FUNCTION_BLOCK "FB_Machine_Spinner"
{ S7_Optimized_Access := 'TRUE' }
VERSION : 0.1
   VAR_INPUT
      Enable : Bool;
      MC_number : Int;
      MC_inRemoteMode : Bool;
      AutoModeFromHandController : Bool;
   END_VAR

   VAR_IN_OUT
      io_in : "UDT_MachineIn";
      io_out : "UDT_MachineOut";
      Status : Int;
      Mode : "UDT_MachineMode";
      cmd : "UDT_CMD";
      order : "UDT_Order";
      pallet : Int;
      fixture : Int;
      ManualVice : Int;
      piecepresent : Array[1..5] of Int;
      viceLocked : Bool;
      viceUnlocked : Bool;
      palletLocked : Bool;
      changePalletReq : Bool;
      lastMission : Int;
      Dispatcher : Array[0..10] of Int;
      subState : Int;
      autoModePrev : Bool;
   END_VAR

   VAR
      "timer" {InstructionName := 'TON_TIME'; LibVersion := '1.0'; S7_SetPoint := 'False'} : Array[0..10] of TON_TIME;
      queryTemp { S7_SetPoint := 'True'} : String;
      doorOpened : Bool;
      enablePrev : Bool;
   END_VAR

   VAR_TEMP
      timeout : Time;
      i : Int;
      countPieces : Int;
      oldStatus : Int;
      tmpUint : UInt;
      Dispatcher_old : Array[0..10] of Int;
   END_VAR


BEGIN
	REGION ENABLE_GATE
	    // Azzero le uscite UNA VOLTA SOLA (fronte di disable) e RETURN.
	    // io_out e' condiviso tra le istanze dei tipi: azzerare a ogni scan
	    // cancellerebbe le uscite mantenute del tipo ATTIVO.
	    IF NOT #Enable THEN
	        IF #enablePrev THEN
	            #io_out.openDoor := FALSE;
	            #io_out.closeDoor := FALSE;
	            #io_out.openVice := FALSE;
	            #io_out.closeVice := FALSE;
	            #io_out.unlockPallet := FALSE;
	            #io_out.lockPallet := FALSE;
	            #io_out.unlockPartOnTable := FALSE;
	            #io_out.lockPartOnTable := FALSE;
	            #io_out.startWork := FALSE;
	            #io_out.startWash := FALSE;
	            #io_out.fuoriIngombro := FALSE;
	        END_IF;
	        #enablePrev := FALSE;
	        RETURN;
	    END_IF;
	    #enablePrev := TRUE;
	END_REGION

	REGION GENERIC_implementation

	    #countPieces := 0;
	    FOR #i := 1 TO 5 DO
	        IF #piecepresent[#i] > 0 THEN
	            #countPieces := #countPieces + 1;
	        END_IF;
	    END_FOR;

	    #oldStatus := #Status;
	    IF #countPieces = 0 THEN
	        IF #pallet = 0 AND #ManualVice = 0 THEN
	            #Status := DINT_TO_INT("UNLOADED");     // totally empty machine
	        ELSE
	            #Status := DINT_TO_INT("EMPTY");        // pallet and fixture mounted on machine but not one piece inside
	        END_IF;

	    ELSIF "DB_Robot".MissionCode = 0 AND #lastMission = "MISSION_LoadPallet_MC" THEN
	        #Status := DINT_TO_INT("EMPTY");
	        #lastMission := 0;

	    ELSIF "DB_Robot".MissionCode = 0 AND #lastMission = "MISSION_UnloadPallet_MC" THEN
	        #Status := DINT_TO_INT("UNLOADED");
	        #lastMission := 0;

	    ELSIF "DB_Robot".MissionCode = 0 AND #lastMission = "MISSION_LoadManVice" THEN
	        #Status := DINT_TO_INT("EMPTY");
	        #lastMission := 0;

	    ELSIF "DB_Robot".MissionCode = 0 AND #lastMission = "MISSION_UnloadManVice" THEN
	        #Status := DINT_TO_INT("UNLOADED");
	        #lastMission := 0;

	    ELSIF FIND(IN1 := "DB_MQTT".lastTopicReceived, IN2 := 'MC1') >= 0 AND #MC_number = 1 THEN  //EG: MC1/CHANGEPALLET
	        IF FIND(IN1 := "DB_MQTT".lastTopicReceived, IN2 := 'CHANGEPALLET') >= 0 THEN
	            #changePalletReq := ("DB_MQTT".lastCmdReceived = 1);
	        ELSIF FIND(IN1 := "DB_MQTT".lastTopicReceived, IN2 := 'CN_STATUS') >= 0 THEN
	            #Status := "DB_MQTT".lastCmdReceived;
	        END_IF;

	    ELSIF FIND(IN1 := "DB_MQTT".lastTopicReceived, IN2 := 'MC2') >= 0 AND #MC_number = 2 THEN  //EG: MC2/CHANGEPALLET
	        IF FIND(IN1 := "DB_MQTT".lastTopicReceived, IN2 := 'CHANGEPALLET') >= 0 THEN
	            #changePalletReq := ("DB_MQTT".lastCmdReceived = 1);
	        ELSIF FIND(IN1 := "DB_MQTT".lastTopicReceived, IN2 := 'CN_STATUS') >= 0 THEN
	            #Status := "DB_MQTT".lastCmdReceived;
	        END_IF;
	    END_IF;

	    IF (#Status >= 0 AND (#Status <> #oldStatus)) THEN
	        "FC_MQTT"(insert := true,
	                  send := false,
	                  topic := CONCAT(IN1 := 'FROM_PLANT/STATUS/MC', IN2 := "INT_TO_STRING_WITHOUT_SIGN"(#MC_number)),
	                  payload := STRING_TO_WSTRING("INT_TO_STRING_WITHOUT_SIGN"(#Status)));
	        #oldStatus := #Status;
	    END_IF;

	END_REGION ;

	FOR #i := 0 TO 10 DO
	    #Dispatcher_old[#i] := #Dispatcher[#i];
	END_FOR;

	REGION Manager CMD from HMI
	    // i comandi HMI non devono interferire col dispatcher
	    IF "DB_MQTT".lastTopicReceived = CONCAT_STRING(IN1 := 'MC', IN2 := "INT_TO_STRING_WITHOUT_SIGN"(#MC_number))
	        AND "DB_RobotMissionStatus".StatusCode = "cmd_waitingNewCmd"
	    THEN
	        IF "DB_MQTT".lastCmdReceived > 0 THEN
	            #cmd.code := "DB_MQTT".lastCmdReceived;
	        END_IF;
	    END_IF;
	END_REGION ;

	REGION Manager MC
	    // Dispatcher COMPLETO (ricetta MQTT -> start fisico -> fine ciclo).

	    // --- Trigger esecuzione query SQL (fuori dal CASE) ---
	    IF #Dispatcher["_master"] >= 10 AND #Dispatcher["_master"] <= 20 THEN
	        "DB_executeQuery"(query := #queryTemp,
	                          exec := #Dispatcher["_master"] = 10);
	    END_IF;

	    CASE #Dispatcher["_master"] OF

	        0:  // IDLE - attesa macchina pronta + robot disponibile, poi pull workorder
	            #cmd.executing := FALSE;
	            #cmd.aborted := FALSE;
	            #io_out.startWork := FALSE;
	            #subState := 0;

	            IF #AutoModeFromHandController
	                AND #io_in.autoMode
	                AND "DB_Robot".MissionCode = 0
	                AND "DB_Robot".Auto
	                AND "DB_Robot".RemoteMode
	                AND #cmd.code <= 0
	                AND "DB_RobotMissionStatus".StatusCode = "cmd_waitingNewCmd"
	            THEN
	                #queryTemp := CONCAT(
	                                     IN1 := 'select top 1 id,PIECE_ID,GRIPPER_ID,MACHINE_ID,PALLET_ID,VICE_ID,QUANTITY,[OPTIONS],Gripper4Pallet,PP_id ',
	                                     IN2 := 'from WORKORDERS where MACHINE_ID=',
	                                     IN3 := "INT_TO_STRING_WITHOUT_SIGN"(#MC_number),
	                                     IN4 := ' AND Status=3 AND PRODUCTED<QUANTITY');
	                #autoModePrev := TRUE;
	                #Dispatcher["_master"] := 10;
	            END_IF;

	        10: // attesa che SQL sia pronto a ricevere
	            IF "DB_executeQuery".readyForNextQuery THEN
	                #Dispatcher["_master"] := 20;
	            END_IF;

	        20: // parsing risultato -> order
	            IF "DB_executeQuery".dataReady AND NOT "DB_executeQuery".dataError THEN
	                #order.ID := "SqlData".data.rows[0].col[0];
	                #order.PIECE := "SqlData".data.rows[0].col[1];
	                #order.GRIPPER := "SqlData".data.rows[0].col[2];
	                #order.MACHINE := "SqlData".data.rows[0].col[3];
	                #order.PALLET := "SqlData".data.rows[0].col[4];
	                #order.VICE := "SqlData".data.rows[0].col[5];
	                #order.QUANTITY := "SqlData".data.rows[0].col[6];
	                #order.OPTION := "SqlData".data.rows[0].col[7];
	                #order.GRIPPER4PALLET := "SqlData".data.rows[0].col[8];
	                #order.PartProgID := "SqlData".data.rows[0].col[9];
	                #order.STATUS := "WORKING";

	                IF #order.ID > 0 THEN
	                    "DB_executeQuery".readyForNextQuery := TRUE;
	                    #queryTemp := '';
	                    #subState := 0;
	                    #Dispatcher["_master"] := 30;
	                END_IF;
	            ELSIF "DB_executeQuery".dataError THEN
	                "DB_executeQuery".readyForNextQuery := TRUE;
	                #Dispatcher["_master"] := 0;
	            END_IF;

	        30: // CHECK PALLET - lancia le missioni; lock/unlock li fa il robot
	            //    via RequestCmd (gestito in SPECIFIC). Solo pallet.
	            CASE #subState OF
	                0:
	                    IF #order.PALLET = #pallet OR #order.PALLET = 0 THEN
	                        #Dispatcher["_master"] := 50;
	                    ELSIF "DB_Robot".MissionCode = 0
	                        AND "DB_RobotMissionStatus".StatusCode = "cmd_waitingNewCmd" THEN
	                        IF #pallet <> 0 THEN
	                            "DB_Robot".MissionCode := "MISSION_UnloadPallet_MC";
	                            "DB_Robot".MCRequested := #MC_number;
	                            #lastMission := "MISSION_UnloadPallet_MC";
	                            #subState := 1;
	                        ELSE
	                            "DB_Robot".MissionCode := "MISSION_LoadPallet_MC";
	                            "DB_Robot".MCRequested := #MC_number;
	                            #lastMission := "MISSION_LoadPallet_MC";
	                            #subState := 2;
	                        END_IF;
	                    END_IF;
	                1: // smontato -> monta il nuovo
	                    IF "DB_Robot".MissionCode = 0
	                        AND "DB_RobotMissionStatus".StatusCode = "cmd_waitingNewCmd" THEN
	                        #pallet := 0;
	                        "DB_Robot".MissionCode := "MISSION_LoadPallet_MC";
	                        "DB_Robot".MCRequested := #MC_number;
	                        #lastMission := "MISSION_LoadPallet_MC";
	                        #subState := 2;
	                    END_IF;
	                2: // montato (robot ha gia' bloccato via RequestCmd) -> prosegui
	                    IF "DB_Robot".MissionCode = 0
	                        AND "DB_RobotMissionStatus".StatusCode = "cmd_waitingNewCmd" THEN
	                        #pallet := DINT_TO_INT(#order.PALLET);
	                        #subState := 0;
	                        #Dispatcher["_master"] := 50;
	                    END_IF;
	            END_CASE;

	            // ---- SERVIZIO ROBOT - logica pinza (fedele al master 100..900) ----

	        50: // (master 100) decisione missione
	            IF "DB_Robot".MissionCode = 0
	                AND "DB_RobotMissionStatus".StatusCode = "cmd_waitingNewCmd"
	                AND "DB_Robot".RemoteMode
	            THEN
	                IF #order.PIECE = 0 THEN
	                    #Dispatcher["_master"] := 58;
	                ELSE
	                    IF #piecepresent[1] = 0 THEN
	                        IF NOT "DB_Robot".GripperOccuped[1] THEN
	                            "DB_Robot".MissionCode := "MISSION_LoadPartOnRobot";
	                            "DB_Robot".GripperRequested := DINT_TO_INT(#order.GRIPPER);
	                            "DB_Robot".MCRequested := #MC_number;
	                            #lastMission := "MISSION_LoadPartOnRobot";
	                            #Dispatcher["_master"] := 51;
	                        ELSE
	                            "DB_Robot".MissionCode := "MISSION_LoadPart_MC";
	                            "DB_Robot".MCRequested := #MC_number;
	                            #lastMission := "MISSION_LoadPart_MC";
	                            #piecepresent[1] := DINT_TO_INT(#order.PIECE);
	                            #Dispatcher["_master"] := 58;
	                        END_IF;
	                    ELSE
	                        IF NOT "DB_Robot".GripperOccuped[1] THEN
	                            IF #order.OPTION.%X0 THEN
	                                // gripper doppio usato singolo
	                                "DB_Robot".MissionCode := "MISSION_UnloadPart_MC";
	                                "DB_Robot".MCRequested := #MC_number;
	                                #lastMission := "MISSION_UnloadPart_MC";
	                                #Dispatcher["_master"] := 52;
	                            ELSE
	                                // gripper doppio usato doppio
	                                "DB_Robot".MissionCode := "MISSION_LoadPartOnRobot";
	                                "DB_Robot".MCRequested := #MC_number;
	                                #lastMission := "MISSION_LoadPartOnRobot";
	                                #Dispatcher["_master"] := 55;
	                            END_IF;
	                        ELSE
	                            IF #order.OPTION.%X0 THEN
	                                #Dispatcher["_master"] := 9999;   // situazione errata
	                            ELSE
	                                "DB_Robot".MissionCode := "MISSION_UnloadPart_MC";
	                                "DB_Robot".MCRequested := #MC_number;
	                                #lastMission := "MISSION_UnloadPart_MC";
	                                #Dispatcher["_master"] := 57;
	                            END_IF;
	                        END_IF;
	                    END_IF;
	                END_IF;
	            END_IF;

	        51: // (master 110) -> rianalizza
	            IF "DB_Robot".MissionCode = 0 THEN
	                #Dispatcher["_master"] := 50;
	            END_IF;

	        52: // (master 150) scarico fatto -> deposita finito a magazzino
	            IF "DB_Robot".MissionCode = 0 THEN
	                #piecepresent[1] := 0;
	                "DB_Robot".MissionCode := "MISSION_UnloadPartFromRobot";
	                #lastMission := "MISSION_UnloadPartFromRobot";
	                #Dispatcher["_master"] := 53;
	            END_IF;

	        53: // (master 160) -> preleva grezzo
	            IF "DB_Robot".MissionCode = 0 THEN
	                "DB_Robot".MissionCode := "MISSION_LoadPartOnRobot";
	                #lastMission := "MISSION_LoadPartOnRobot";
	                #Dispatcher["_master"] := 54;
	            END_IF;

	        54: // (master 170) -> preleva secondo grezzo, poi rianalizza
	            IF "DB_Robot".MissionCode = 0 THEN
	                "DB_Robot".MissionCode := "MISSION_LoadPartOnRobot";
	                #lastMission := "MISSION_LoadPartOnRobot";
	                #Dispatcher["_master"] := 50;
	            END_IF;

	        55: // (master 200) grezzo in pinza -> scarica finito dalla macchina
	            IF "DB_Robot".MissionCode = 0 THEN
	                "DB_Robot".MissionCode := "MISSION_UnloadPart_MC";
	                "DB_Robot".MCRequested := #MC_number;
	                #lastMission := "MISSION_UnloadPart_MC";
	                #Dispatcher["_master"] := 56;
	            END_IF;

	        56: // (master 210) -> rianalizza
	            IF "DB_Robot".MissionCode = 0 THEN
	                #piecepresent[1] := 0;
	                #Dispatcher["_master"] := 50;
	            END_IF;

	        57: // (master 300) finito scaricato -> inserisci grezzo in macchina
	            IF "DB_Robot".MissionCode = 0 THEN
	                "DB_Robot".MissionCode := "MISSION_LoadPart_MC";
	                "DB_Robot".MCRequested := #MC_number;
	                #lastMission := "MISSION_LoadPart_MC";
	                #piecepresent[1] := DINT_TO_INT(#order.PIECE);
	                #Dispatcher["_master"] := 58;
	            END_IF;

	        58: // (master 900) macchina pronta: deposita finito ancora in pinza, poi RICETTA
	            IF "DB_Robot".MissionCode = 0
	                AND (#order.PALLET = #pallet OR #order.PALLET = 0)
	                AND #order.PIECE = #piecepresent[1]
	            THEN
	                IF "DB_Robot".GripperOccuped[1] OR "DB_Robot".GripperOccuped[2] THEN
	                    "DB_Robot".MissionCode := "MISSION_UnloadPartFromRobot";   // Robot -> TRAY
	                    #lastMission := "MISSION_UnloadPartFromRobot";
	                ELSE
	                    #Dispatcher["_master"] := 90;
	                END_IF;
	            END_IF;

	            // ---- SEQUENZA CICLO: ricetta -> start -> fine ciclo -> cycle done ----

	        90: // DISPATCH RICETTA - setMacro #10200 = PartProgID
	            "FC_MQTT"(insert := TRUE,
	                      send := FALSE,
	                      topic := CONCAT(IN1 := 'FROM_PLANT/HAAS_CMD/MC',
	                                      IN2 := "INT_TO_STRING_WITHOUT_SIGN"(#MC_number)),
	                      payload := STRING_TO_WSTRING(CONCAT(
	                                                                                       IN1 := '{"cmd":"setMacro","var":10200,"value":',
	                                                                                       IN2 := DINT_TO_STRING(#order.PartProgID),
	                                                                                       IN3 := '}')));
	            #timer[1](IN := TRUE,
	                      PT := T#10s);
	            #Dispatcher["_master"] := 91;

	        91: // attesa esito ricetta: ACK -> ok ; NACK -> fallita
	            IF "DB_MQTT".lastTopicReceived
	                = CONCAT(IN1 := 'HAAS_ACK/MC',
	                         IN2 := "INT_TO_STRING_WITHOUT_SIGN"(#MC_number))
	            THEN
	                #timer[1](IN := FALSE,
	                          PT := T#10s);
	                #Dispatcher["_master"] := 92;
	            ELSIF "DB_MQTT".lastTopicReceived
	                = CONCAT(IN1 := 'HAAS_NACK/MC',
	                         IN2 := "INT_TO_STRING_WITHOUT_SIGN"(#MC_number))
	            THEN
	                #timer[1](IN := FALSE,
	                          PT := T#10s);
	                #Dispatcher["_master"] := 9999;
	            ELSIF #timer[1].Q THEN
	                #timer[1](IN := FALSE,
	                          PT := T#10s);
	                #Dispatcher["_master"] := 9999;
	            END_IF;

	        92: // START - Q_startWork alto fino a caduta AutoMode (robot fuori ingombro)
	            IF #io_out.fuoriIngombro THEN
	                #io_out.startWork := TRUE;
	                #timer[6](IN := TRUE,
	                          PT := T#30s);   // safety conta solo da quando do lo start
	                IF #timer[6].Q THEN
	                    #io_out.startWork := FALSE;
	                    #timer[6](IN := FALSE,
	                              PT := T#30s);
	                    #Dispatcher["_master"] := 9999;
	                END_IF;
	            END_IF;
	            IF NOT #io_in.autoMode THEN
	                #io_out.startWork := FALSE;
	                #autoModePrev := FALSE;
	                #timer[6](IN := FALSE,
	                          PT := T#30s);
	                #Dispatcher["_master"] := 95;
	            END_IF;

	        95: // attesa fine ciclo - AutoMode torna alto (M30)
	            IF #io_in.autoMode AND NOT #autoModePrev THEN
	                #autoModePrev := TRUE;
	                #Dispatcher["_master"] := 100;
	            END_IF;
	            IF #io_in.autoMode THEN
	                #autoModePrev := TRUE;
	            END_IF;

	        100: // CYCLE_DONE - notifica backend (incrementa PRODUCTED)
	            "FC_MQTT"(insert := TRUE,
	                      send := FALSE,
	                      topic := CONCAT(IN1 := 'FROM_PLANT/CYCLE_DONE/MC',
	                                      IN2 := "INT_TO_STRING_WITHOUT_SIGN"(#MC_number)),
	                      payload := STRING_TO_WSTRING(DINT_TO_STRING(#order.ID)));
	            "FC_MQTT"(insert := TRUE,
	                      send := FALSE,
	                      topic := CONCAT(IN1 := 'FROM_PLANT/STATUS/MC',
	                                      IN2 := "INT_TO_STRING_WITHOUT_SIGN"(#MC_number)),
	                      payload := STRING_TO_WSTRING('CYCLE_COMPLETED'));
	            #Dispatcher["_master"] := 0;

	        9999: // ERROR - reset via MQTT "MC_resetError" dall'HMI
	            IF "DB_MQTT".lastTopicReceived
	                = CONCAT(IN1 := 'MC', IN2 := "INT_TO_STRING_WITHOUT_SIGN"(#MC_number))
	                AND "DB_MQTT".lastCmdReceived = "MC_resetError"
	            THEN
	                #Dispatcher["_master"] := 0;
	                #Status := DINT_TO_INT("UNLOADED");
	                #cmd.code := 0;
	                #cmd.executing := FALSE;
	                #cmd.aborted := FALSE;
	                #order.ID := 0;
	                #order.PIECE := 0;
	                #lastMission := 0;
	                #subState := 0;
	                #io_out.startWork := FALSE;
	                "FC_MQTT"(insert := TRUE,
	                          send := FALSE,
	                          topic := CONCAT(IN1 := 'FROM_PLANT/STATUS/MC',
	                                          IN2 := "INT_TO_STRING_WITHOUT_SIGN"(#MC_number)),
	                          payload := STRING_TO_WSTRING("INT_TO_STRING_WITHOUT_SIGN"(#Status)));
	            END_IF;

	    END_CASE;

	    // Fuori ingombro robot: alto quando il robot NON sta servendo questa MC
	    #io_out.fuoriIngombro := ("DB_Robot".MCRequested <> #MC_number);
	END_REGION

	REGION Update HMI
	    //Dispatchers value
	    FOR #i := 0 TO 10 DO
	        IF #Dispatcher_old[#i] <> #Dispatcher[#i] THEN
	            "FC_MQTT"(insert := true,
	                      send := false,
	                      topic := CONCAT(IN1 := 'FROM_PLANT/DISPATCH/MC', IN2 := "INT_TO_STRING_WITHOUT_SIGN"(#MC_number), IN3 := '/', IN4 := "INT_TO_STRING_WITHOUT_SIGN"(#i)),
	                      payload := STRING_TO_WSTRING("INT_TO_STRING_WITHOUT_SIGN"(#Dispatcher[#i])));

	            #Dispatcher_old[#i] := #Dispatcher[#i];
	        END_IF;
	    END_FOR;
	END_REGION ;

	REGION Management cmd from robot to MC
	    IF #Status <> "MANUAL"
	        AND "DB_Robot".MCRequested = #MC_number
	        AND NOT #cmd.executing
	        AND #cmd.code = 0 THEN

	        IF "DB_RobotMissionStatus".RequestCmd.Lock_Pallet THEN
	            #cmd.code := "MC_lockPallet";
	        ELSIF "DB_RobotMissionStatus".RequestCmd.Unlock_Pallet THEN
	            #cmd.code := "MC_unlockPallet";

	        ELSIF "DB_RobotMissionStatus".RequestCmd.Lock_Vice THEN
	            #cmd.code := "MC_closeVice";
	        ELSIF "DB_RobotMissionStatus".RequestCmd.Unlock_Vice THEN
	            #cmd.code := "MC_openVice";

	        ELSIF "DB_RobotMissionStatus".RequestCmd.Open_door THEN
	            #cmd.code := "MC_openDoor";
	        ELSIF "DB_RobotMissionStatus".RequestCmd.Close_door THEN
	            #cmd.code := "MC_closeDoor";

	        ELSIF "DB_RobotMissionStatus".RequestCmd.Lock_partOnTable THEN
	            #cmd.code := "MC_lockPartOnTable";
	        ELSIF "DB_RobotMissionStatus".RequestCmd.Unlock_partOnTable THEN
	            #cmd.code := "MC_unlockPartOnTable";
	        END_IF;
	    END_IF;
	END_REGION

	REGION SPECIFIC_implementation
	    // SPINNER: porta PILOTATA dal PLC (Q_openDoor/Q_closeDoor).
	    // MC_startWork = no-op (lo start fisico lo fa il dispatcher @ stato 92).
	    CASE #cmd.code OF
	        "MC_openVice":
	            #timeout := T#1s;
	            #io_out.openVice := TRUE;
	            #io_out.closeVice := FALSE;
	            #cmd.executing := TRUE;
	        "MC_closeVice":
	            #timeout := T#1s;
	            #io_out.openVice := FALSE;
	            #io_out.closeVice := TRUE;
	            #cmd.executing := TRUE;
	        "MC_unlockPallet":
	            #timeout := T#5s;
	            #io_out.unlockPallet := TRUE;
	            #io_out.lockPallet := FALSE;
	            #cmd.executing := TRUE;
	        "MC_lockPallet":
	            #timeout := T#5s;
	            #io_out.unlockPallet := FALSE;
	            #io_out.lockPallet := TRUE;
	            #cmd.executing := TRUE;
	        "MC_openDoor":
	            // Spinner: uscita porta SINGOLA mantenuta. Apre = Q_openDoor TRUE.
	            #timeout := T#5s;
	            #io_out.openDoor := TRUE;
	            #cmd.executing := NOT #io_in.doorOpened;   // confermato dal feedback "aperta"
	        "MC_closeDoor":
	            // Spinner: chiude togliendo l'uscita. Nessun feedback "chiusa": solo timeout.
	            #timeout := T#5s;
	            #io_out.openDoor := FALSE;
	            #cmd.executing := TRUE;
	        "MC_lockPartOnTable":
	            #timeout := T#1s;
	            #io_out.lockPartOnTable := TRUE;
	            #io_out.unlockPartOnTable := FALSE;
	            #cmd.executing := TRUE;
	        "MC_unlockPartOnTable":
	            #timeout := T#1s;
	            #io_out.lockPartOnTable := FALSE;
	            #io_out.unlockPartOnTable := TRUE;
	            #cmd.executing := TRUE;
	        "MC_startWork":
	            // start gestito dal dispatcher (stato 92): qui no-op
	            #timeout := T#30s;
	            #cmd.executing := TRUE;
	        ELSE
	            //unknown command
	            #cmd.aborted := TRUE;
	            #cmd.executing := FALSE;
	            #cmd.executed := FALSE;
	    END_CASE;

	    #timer[0](IN := #cmd.executing,
	              PT := #timeout);

	    IF (#timer[0].Q) THEN
	        #cmd.executing := FALSE;
	    END_IF;

	    #cmd.executed := NOT (#cmd.executing);
	    #cmd.aborted := NOT (#cmd.executing) AND NOT (#cmd.executed);

	    IF #cmd.code = "MC_unlockPallet" AND (#cmd.executed OR #io_in.palletUnlocked) THEN
	        #palletLocked := false;
	    END_IF;
	    IF #cmd.code = "MC_lockPallet" AND (#cmd.executed OR NOT #io_in.palletUnlocked) THEN
	        #palletLocked := true;
	    END_IF;

	    IF #cmd.code = "MC_openVice" AND (#cmd.executed OR #io_in.viceOpened) THEN
	        #viceLocked := false;
	    END_IF;
	    IF #cmd.code = "MC_closeVice" AND (#cmd.executed OR NOT #io_in.viceOpened) THEN
	        #viceLocked := true;
	    END_IF;

	    IF #cmd.executed THEN
	        #cmd.code := 0;
	    END_IF;

	END_REGION ;
END_FUNCTION_BLOCK

